INTERFACE I_SEW_Movisafe

PROPERTY bSTO : BOOL
GET
END_GET
END_PROPERTY

END_INTERFACE

(* stored: Version 1.1.0.1, ProductVersion 3.1.4024.12
   Itf I_SEW_Movisafe: Id {4d308d10-7209-0ca2-12b5-dec8b03abd5f}
   Property bSTO: Id {2d79631d-512f-06ef-3d6e-7e1fbd71b292}
   Get Get: Id {2f80e9c7-6ce0-08ab-245c-5c74e93d0656} *)
